{attribute 'qualified_only'}
VAR_GLOBAL
END_VAR

(* stored: Version 1.1.0.1
   GVL GVL_PLC_Interfances: Id {6a6e2e4e-a4f2-497a-9e06-56d7bc60be59} *)
